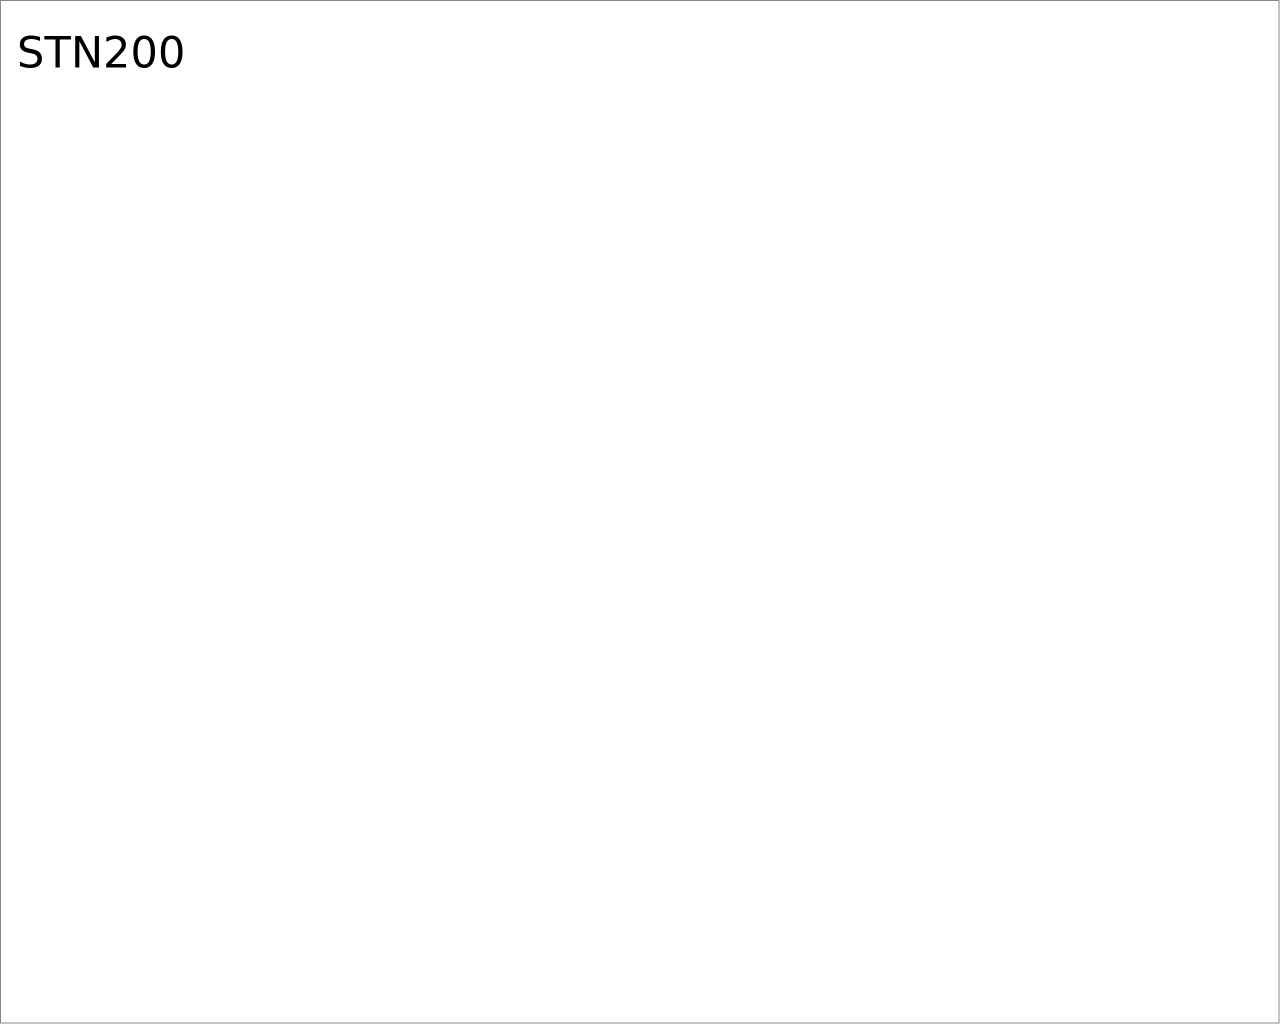
VISUALIZATION Visualization  // 1280x1024
    Label (-12,4 227x97), "STN200"
END_VISUALIZATION

(* stored: Version 1.1.0.1, ProductVersion 3.1.4024.2
   Visu Visualization: Id {c34c3bce-33f5-4345-a93e-f997e55115a3} *)
